ABB RobotStudio station: Tp1_20201208-212119.rsstn

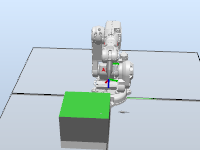
Station Tp1 (saved by RobotStudio 20.2.9116.0)
Controller IRB_140_6kg_0.81m
  mechanical unit ROB_1: IRB140_6_81_C_03, 6 joints, base frame (0, 0, 0) mm
Layout (positions relative to the parent item):
  - IRB140_6_81_C_03 [mechanism, from Robots\IRB140_6_81_C_G_03.rslib] at (0, 0, 0) mm; joint values [-0.7166, 0.5968, -0.2821, -0.054, 0.5236, 0] (rad or m)
  - Mesa [part]
  - Perno [part]
  - Pinza [mechanism] at (506.29, 0, 679.5) mm, rotated rx 180 ry 60 rz 180 deg
      TCP Pinza at (0, 0, 137) mm, rotated rx 0 ry 0 rz -22.5 deg
      links: Dummy
Attachment: Pinza is attached to IRB140_6_81_C_03 / Link6
EventTableEntry 1017: Group=, Trigger=DO_Pinza 1018, Actions=[EventTableActionAttach 1019], Comment=, ActivationMode=2, Cyclic=false
EventTableTriggerIO 1018: IOValue=[1], IRC5Controller=? -1, Operator=0, SignalSource=IRB_140_6kg_0.81m 515
EventTableActionAttach 1019: AttachmentParent=Pinza 1013, AttachmentChild=Perno 1009, MountObject=false, Offset=[X=1, Y=0, Z=0, W=0, X=0, Y=1, Z=0, W=0, X=0, Y=0, Z=1, W=0, X=0, Y=0, Z=0, W=1], FlangeIndext=0, FindNearest=false
EventTableEntry 1020: Group=, Trigger=DO_Pinza 1021, Actions=[EventTableActionDetach 1022], Comment=, ActivationMode=2, Cyclic=false
EventTableTriggerIO 1021: IOValue=[0], IRC5Controller=? -1, Operator=0, SignalSource=IRB_140_6kg_0.81m 515
EventTableActionDetach 1022: AttachmentParent=Pinza 1013, AttachmentChild=Perno 1009
Collision set Colision Perno- Mesa: Perno against Mesa, near miss 0.02 m
Collision set Colision Robot - Mesa: IRB140_6_81_C_03 against Mesa, near miss 0 m
Collision set Colision Pinza - Mesa: Mesa against Pinza, near miss 0 m
Targets, tools, work objects and paths stored in the station, written as RAPID:
! task T_ROB1
MODULE CalibData
  PERS tooldata Pinza:=[TRUE,[[0,0,137],[0.98078528,0,0,-0.195090322]],[0.5,[0,0,100],[1,0,0,0],0,0,0]];
ENDMODULE

